(* CODESYS project set_in_mode.20190528.1.project

Project tree, tasks and I/O mapping:
  MIC7001 : Changsha Xiangji-ARM Cortex A9(xilinx zynq7000)-linux, Changsha Xiangji Hiden Technology Co.Ltd, version 3.5.10.40
    application Application
      libraries: Standard, * (System); CAA File, * (CAA Technical Workgroup); CAA Types Extern, * (CAA Technical Workgroup); CAA Callback Extern, * (CAA Technical Workgroup); SysMem, * (System); Util, 3.5.11.0 (System); SysFile, 3.5.9.0 (System); SysTypes Interfaces, * (System); CAN API, 1.0.0.3 (3S - Smart Software Solutions GmbH); SysTime, * (System); CAA DTUtil Extern, 3.5.12.0 (CAA Technical Workgroup); CAA SerialCom, 3.5.12.0 (CAA Technical Workgroup); cyber gpio, 3.5.10.40 (cyber); AC_DataLog, 3.5.13.0 (3S - Smart Software Solutions GmbH)
      task MainTask (cyclic, interval 20 ms, priority 15) calls prg_set_inmode
      program prg_set_inmode [ST]
      functions/
        function fn_write_in_mode_file [ST]
        function fn_read_in_mode_file [ST]
    SoftMotion General Axis Pool
  text list GlobalTextList
*)

// MIC7001/Application/prg_set_inmode
PROGRAM prg_set_inmode
VAR
	stat:UINT := 0;
	old_in_mode:ARRAY[0..47] OF UINT;  //从已有文件中读出的配置
	in_mode:ARRAY[0..47] OF UINT;   //当前设定的配置
	number :UINT := 48;  //通道总数
	i: UINT;
	inmode_file:STRING:='in_mode.txt';
	
	MODE_0_5V :UINT := 0;
	MODE_0_36V :UINT := 1;
	MODE_0_20mA :UINT := 2;
	MODE_0_30Kohm :UINT := 3;
	MODE_DI_HIGH :UINT := 4;
	MODE_DI_LOW :UINT := 5;
END_VAR


CASE stat OF
0: //read inmode.txt
	IF fn_read_in_mode_file(pInMOde := ADR(old_in_mode), number := number) THEN
		stat := 50;
	ELSE 
		stat := 10;
	END_IF
10: //need write
	IF fn_write_in_mode_file(pInMode := ADR(in_mode), number := number) THEN
		stat := 100; //succeed
	END_IF

50: //the file inmode.txt is exist.
	FOR i := 0 TO number-1 DO
		IF old_in_mode[i] <> in_mode[i] THEN
			stat := 10; //write new config
			RETURN;
		END_IF
	END_FOR
	stat := 100;

100: //succeed, return;
	RETURN;
END_CASE

//默认全部设置为  0~5V输入
FOR  i := 0 TO number-1 DO
	in_mode[i] := 0;
END_FOR

//            上面的代码不用改动
//*********************************************************


//根据实际情况设置每个端口的类型
in_mode[0] := MODE_0_20mA;  //0~20 mA 
//in_mode[1] := MODE_0_5V;  //默认为  MODE_0_5V， 可以不设置
in_mode[2] := MODE_0_36V;  
in_mode[3] := MODE_0_36V;
//.........
in_mode[47] := MODE_DI_LOW;   //最后一个

END_PROGRAM

// MIC7001/Application/functions/fn_read_in_mode_file
FUNCTION fn_read_in_mode_file : BOOL
VAR_INPUT
	pInMode :POINTER TO UINT;
	number:UINT;
END_VAR
VAR
	hFile: RTS_IEC_HANDLE;
	udiOpenError: RTS_IEC_RESULT;
	udiReadError: RTS_IEC_RESULT;
	i :DWORD;
	iTemp: UDINT;
	udiPos: UDINT;
	str: STRING(65535);
	str_size: __XWORD;
	udiByteRead: LWORD;

	len_of_line: INT;
	len_of_number :INT;
	magicNumber:REAL;
	check_sum:REAL:= 0;
	temp_num:REAL;
	index :UINT;
	mode: UINT;
END_VAR

fn_read_in_mode_file := FALSE;

//检测文件是否存在
hFile := sysfileopen(szFile := prg_set_inmode.inmode_file, am := sysfile.AM_READ, pResult:= ADR(udiOpenError));
IF hFile = RTS_INVALID_HANDLE	THEN  //文件不存在
	RETURN;
END_IF

//文件存在，开始读取内容
udiPos := SysFileSetPos(hFile:=hFile, ulOffset := 0);
udiByteRead := sysfile.SysFileRead(hfile := hFile,pbyBuffer := ADR(str), ulSize := SIZEOF(str), pResult := ADR(udiReadError));
IF udiByteRead < 1 THEN  //读取失败
	sysfile.SysFileClose(hFile := hFile);
	RETURN;
END_IF
sysfile.SysFileClose(hFile);

//读取本行的数字
FOR i := 0 TO number-1 DO
	len_of_number := find(str, '$N');
	mode := STRING_TO_UINT(left(str,len_of_number-1));
	str := delete(str, len_of_number,1);	
	pInMode[i] := mode;
END_FOR

fn_read_in_mode_file := TRUE;
RETURN;

END_FUNCTION

// MIC7001/Application/functions/fn_write_in_mode_file
FUNCTION fn_write_in_mode_file : BOOL
VAR_INPUT
	pInMode :POINTER TO UINT;
	number:UINT;
END_VAR
VAR
	bak_file_prefix:STRING :=ANY_TO_STRING("in_mode_bak_");
	bak_file:STRING := ANY_TO_STRING("");	
	hFile: RTS_IEC_HANDLE;
	udiDeleteError: RTS_IEC_RESULT;
	udiOpenError: RTS_IEC_RESULT;
	udiWriteError: RTS_IEC_RESULT;
	filesize: __XWORD;
	i :DWORD;
	iTemp: UDINT;
	udiPos: UDINT;
	str: STRING(256);
	str_size: __XWORD;
	udiByteWrite: LWORD;
	check_sum:REAL := 0;
END_VAR

fn_write_in_mode_file := FALSE;

IF number = 0 THEN
	RETURN;
END_IF

hFile := sysfileopen(szFile := prg_set_inmode.inmode_file, am := sysfile.AM_WRITE, pResult := ADR(udiOpenError));
IF hFile = RTS_INVALID_HANDLE THEN //创建文件失败
	RETURN;
END_IF
	
udiPos := SysFileSetPos(hFile:=hFile, ulOffset:=0);	
str:= ANY_TO_STRING('');
FOR i := 0 TO number-1 DO
	str := concat(str, ANY_TO_STRING(pInMode[i]));
	str := concat(str, '$N');	
END_FOR

str_size := ANY_TO_DWORD(len(str));
udiByteWrite := sysfile.SysFileWrite(hFile := hFile,pbyBuffer := ADR(str),ulSize := str_size, pResult := ADR(udiWriteError));

sysfile.SysFileClose(hFile);
fn_write_in_mode_file := TRUE;

END_FUNCTION
